{attribute 'qualified_only'}
VAR_GLOBAL
END_VAR

(* stored: Version 1.1.0.1, ProductVersion 3.1.4022.7
   GVL GVL_06_Output_Servo_Motor_Robot: Id {0667a752-89ca-42b3-9a32-56d2c674872f} *)
